//variables must be referenced GVL_MOTION.etc b/c of attribute
//persistent data causes problems when changing variable declarations
{attribute 'qualified_only'}
VAR_GLOBAL
	//motor control signals
	
	xCon					:CTR_SIGNALS_INTERNAL;
	xcCon					:CTR_SIGNALS_INTERNAL;
	yCon					:CTR_SIGNALS_INTERNAL;
	zCon					:CTR_SIGNALS_INTERNAL;
	
	xJogFW					:BOOL;
	xJogBW					:BOOL;
	yJogFW					:BOOL;
	yJogBW					:BOOL;
	zJogFW					:BOOL;
	zJogBW					:BOOL;
	
	MOVEXYZ					:BOOL;
	
	ED2008O AT %Q*			:ED2008_46D0FC69;
	Z_BRAKE_OFF				:BOOL;
	
	//external controls
	STOP_EXT				:BOOL;
	STOP_INT				:BOOL; //control signal
	EXT_CTR					:MOTION_CTR; 
	TEST_CTR				:MOTION_CTR; //test buffer for MQTT
	HB						:HB;
	{attribute 'TcEncoding':='UTF-8'}
	TopicRcv				:STRING(255); //for MQTT
	
	//script variables
	
	InstructionBuffer		:MOTION_INSTRUCTION; //set externally (MQTT) or locally
	TestBuffer				:MOTION_INSTRUCTION; //test buffer for MQTT
	EmptyInstruction		:MOTION_INSTRUCTION;
	Script 					:ARRAY[0..99] OF MOTION_INSTRUCTION; //add commands from instruction buffer or load script
	ScriptReadBuffer		:ARRAY[0..99] OF MOTION_INSTRUCTION; //buffer for ScriptRead
	ContinuousMode			:BOOL; //override number of script runs and run until set false
	ScriptEnd				:INT						:= 0; //empty/not executed
	InstructionState		:INT						:= 0; //control case statement in RunCommands
	TxtBxWaitOK				:BOOL						:= TRUE; //hide text box
	HaltMem					:BOOL						:= FALSE; //part of the waitOK motion button control
	
	
	STATUS					:STATUS;
	ActiveBasin				:BASIN;
	BasinA					:BASIN	:= (Name := 'BasinA',
										xMin := 0,			
										xMax := 100000,
										yMin := 0,
										yMax := 5000);
	
	BasinB					:BASIN	:= (Name := 'BasinB',
										xMin := 0,			
										xMax := 100000,
										yMin := 5050,
										yMax := 8991);
	BASINLAMPA				:BOOL;
	BASINLAMPB				:BOOL;
	CSV_ROW					:INT						:= 0;
	
	//variables for script list
	
	LISTSTART				:BOOL						:= FALSE;
	LISTEND					:BOOL						:= FALSE;
	LIST					:ARRAY[0..999] OF T_MaxString;
	LISTCNT					:INT						:= 0;
	SCRIPTNAME				:SCRIPTNAME;
	
	//filelistp				:VISU_FBFileListProvider;
	
	xOut					:OUT_SIGNALS;
	xCOut					:OUT_SIGNALS;
	yOut					:OUT_SIGNALS;	
	zOut					:OUT_SIGNALS;
	xHomeStatus				:MOTION_FB_STATUS;
	xCHomeStatus			:MOTION_FB_STATUS;
	yHomeStatus				:MOTION_FB_STATUS;
	zHomeStatus				:MOTION_FB_STATUS;
	
	CurInstruction			:INT						:= 0; //current instruction
	NextInstruction			:INT; //only for display
	RUN_INDEX				:INT						:= 1; //increment after script run
	
	//for the drop down lists
	
	xyzCMDSelect			:ARRAY[0..4] OF MotionType	:= [0,1,2,3,4];
	
	//safety controls

	zSafeSet				:BOOL						:= FALSE;
	zSafeDisable			:BOOL						:= FALSE; 	(*in zAxisMoreLogic*)
	zSafePosition			:LREAL						:= 0;	
	
	//homing variables
	
	HomingState				:INT						:= 0;
	RevCouplePrep			:BOOL						:= FALSE;
	//x and y stage from rail to top of y stage
	//z stage from rail to bottom of z stage
	CARRIAGE_OFFSETS		:ARRAY[0..2] OF LREAL		:= [500,250,100]; //also in STATUS
END_VAR

VAR_GLOBAL
	AxesLocated				:BOOL						:= FALSE;
	xLocated				:BOOL						:= FALSE;
	yLocated				:BOOL						:= FALSE;
	zLocated				:BOOL						:= FALSE;
							
END_VAR

(* stored: Version 1.1.0.1, ProductVersion 3.1.4026.18
   GVL GVL_MOTION: Id {ea33deb8-8627-4a0d-a3f0-288faa3aa9d9} *)
